TYPE VisuStructPoint :
STRUCT
	iX: INT;
	iY: INT;
END_STRUCT
END_TYPE

(* stored: Version 1.1.0.1, ProductVersion 3.1.4024.2
   DUT VisuStructPoint: Id {367ee55d-3662-448a-bf5e-dd2ff10b2cc1} *)
